// Brief: Slave Arm Adjust
FUNCTION_BLOCK PUBLIC FB_SlaveCtrlOffScreenTest EXTENDS FB_SlaveCtrlAdjust
VAR CONSTANT
	m_sampleNum :INT := 9;
END_VAR
VAR
	// sample joint position 
	m_sampleSetupJntPos :ARRAY[1..m_sampleNum] OF Vec5d;
	m_sampleSlaveJntPos :ARRAY[1..m_sampleNum] OF Vec6d;
	
	// sample signal
	m_sampleSignal : FB_AdjustLongPress;
	
	// current sample number
	m_curSampleNum :INT := 0;
	
	m_logStr:STRING;
	m_armStr:STRING;
	
	idx:INT:=0;
END_VAR

// override this function in each exact controller
METHOD PROTECTED calcCmdJntPos : BOOL
VAR_IN_OUT CONSTANT
	i_endoscopePose : ST_Frame;
	i_masterStatus :ST_MasterStatus;
	i_setupStatus: ST_SetupStatus;
	i_slaveArm :FB_SlaveArm;
END_VAR
VAR
	i:INT;
END_VAR
SUPER^.calcCmdJntPos(i_endoscopePose,i_masterStatus, i_setupStatus, i_slaveArm);

IF m_curSampleNum > m_sampleNum THEN
	m_isFinished :=TRUE;
	AGILOG_DebugStop();
	g_offScreenTest.m_enterOffScreenTestMode[idx] := FALSE;
	RETURN;
END_IF


IF i_slaveArm.adjustOn THEN //After pressing the button, the joint is enabled.
	FOR i:=1 TO 3 DO
		m_jntEnableFlag[i] := 1;
		m_jntOPMode[i] := DriverOPMode_Trq;//current joint enter adjust mode
		m_cmdJntPos[i] := i_slaveArm.curJntPos[i];
	END_FOR
END_IF	
				
	
IF g_offScreenTest.m_dataRecordFlag[idx] THEN
	g_offScreenTest.m_caliPointStartFlag[m_curSampleNum] := FALSE;//the last point finish
	g_offScreenTest.m_caliPointEndFlag[m_curSampleNum] := TRUE;
	
	m_curSampleNum := m_curSampleNum +1;
		
	m_sampleSetupJntPos[m_curSampleNum] := SetupArmControl.m_setupRobot.m_setupArms[i_slaveArm.armIdx].curJntPos;
	m_sampleSlaveJntPos[m_curSampleNum] := i_slaveArm.curDHJntPos;
	
	AGILOG_DEBUG(m_armStr, FALSE, 1);
	
//	AGILOG_DEBUG(SetupArmControl.m_setupRobot.m_setupArms[i_slaveArm.armIdx].curJntPos, FALSE, 2);
//	AGILOG_DEBUG(i_slaveArm.curDHJntPos, FALSE, 1);
	
	AGILOG_DEBUG(RobotDynamics.m_instruViewCheck.m_instruPoseInScope[i_slaveArm.armIdx].m_pos,FALSE, 1);
	
	g_offScreenTest.m_caliPointStartFlag[m_curSampleNum] := TRUE;//the next point begin
	g_offScreenTest.m_caliPointEndFlag[m_curSampleNum] := FALSE;
END_IF
END_METHOD

METHOD PUBLIC Init : BOOL
VAR_IN_OUT CONSTANT
	i_slaveArm	:FB_SlaveArm;
END_VAR
VAR_IN_OUT 
	r_slaveArmCtrlCmd :ST_SlaveArmCtrlCmds;
END_VAR

VAR
	fileName:STRING;
END_VAR
//init
SUPER^.Init(i_slaveArm,r_slaveArmCtrlCmd);
m_jntEnableFlag :=g_zeroVec8i;

idx:=i_slaveArm.armIdx;
g_offScreenTest.m_dataRecordCount[idx]:=0;

m_curSampleNum:=1;
 
fileName := CONCAT('OffScreenCali_arm', INT_TO_STRING(i_slaveArm.armIdx));
fileName := CONCAT(fileName, '.txt');
AGILOG_DebugStart(fileName);

m_logStr := '########Start Off-screen calibration sampling.########';
AGILOG_DEBUG(m_logStr, TRUE, 1);

m_armStr := concat('slaveArm', INT_TO_STRING(i_slaveArm.armIdx));
END_METHOD

END_FUNCTION_BLOCK

(* stored: Version 1.1.0.1, ProductVersion 3.1.4024.11
   POU FB_SlaveCtrlOffScreenTest: Id {0de35542-f418-484a-8b25-3d2d3fcee84c}, SpecialFunc None
   Method calcCmdJntPos: Id {281a553a-abc7-436e-8e20-e6db994ac83e}
   Method Init: Id {e01a414e-349a-49ce-840c-54e7ef82b96a} *)
